Fanuc KAREL source: kt00177.KL

-- PROVISIONAL review KL for V1013-1; original PC SHA256 16e69875a06ac2ecdefd8594f0ce1c6cd54c1910b775416597ce470e5432d911
-- Incomplete behavior may be omitted. Consult companion uncertainty JSON. Do not deploy.
PROGRAM KT00177
%NOLOCKGROUP
VAR
  I2 : INTEGER
  OUT : INTEGER
-- UNRESOLVED_DECL Y1 type=002018
BEGIN
  -- UNRESOLVED_PC offsets 5-19; opcodes 2E,22,9D,33,B2
  -- UNRESOLVED_PC offsets 24-35; opcodes 2E,23
  -- UNRESOLVED_PC offsets 40-62; opcodes 22,9D,33,B1,21,56,23
  -- UNRESOLVED_PC offsets 67-71; opcodes 7F
END KT00177
